# EPICS autosave request: iocBoot/sioc-asta-pv05/pv.req
file ../pvCommon.req P=$(P)
file ../scanPv.req P=$(P)
$(P):SCAN:SSBEAM
$(P):SCAN:SSBEAMPUMP
$(P):Z:LOCK:ENABLE
$(P):Z:LOCK:SLOPE
$(P):Z:LOCK:INT
$(P):GRABIMAGES:NSTATIC
$(P):GRABIMAGES:NBG
$(P):GRABIMAGES:SSTRIGMODE
$(P):GRABIMAGES:I0ENABLE
$(P):MULTISTATIC:ENABLE
